PROGRAM ReadCP67
VAR
	
	ReadActLightLvlBoardroom :FB_DALIV2QueryActualLevel;  //Used to read back actual light lvl to correct dimmer on CP67 ask Plug top


	ADS_READ:ADSREAD;
	
	ADX_READ_DMXR:ADSREAD;
	ADX_READ_DMXG:ADSREAD;
	ADX_READ_DMXB:ADSREAD;
	
	DMX_Enable_READ:ADSREAD;
	
	HoldCP67BoardRoomLightsOn:BYTE;
	

	Sample		: BYTE;
	
	DMXRValues	:	ARRAY [0..7] OF BYTE;
	DMXGValues	:	ARRAY [0..7] OF BYTE;
	DMXBValues	:	ARRAY [0..7] OF BYTE;
	
	CP67_DMX_Enable	:	BOOL;
	
	FBDALIV2Dimmer1Switch : ARRAY [1..15] OF FB_DALIV2Dimmer1Switch;
	CASECP67BoardRoomLightsOn : INT;

END_VAR

sample := sample + 1;

FBDALIV2Dimmer1Switch[1](stCommandBuffer:= stCommandBuffer);
FBDALIV2Dimmer1Switch[2](stCommandBuffer:= stCommandBuffer);
ReadActLightLvlBoardroom(stCommandBuffer := stCommandBuffer , nActualLevel => BoardroomActualLightLvl ); 

IF CP67BoardRoomLightsOn <> HoldCP67BoardRoomLightsOn THEN
HoldCP67BoardRoomLightsOn := CP67BoardRoomLightsOn;
CASECP67BoardRoomLightsOn := 10;
END_IF

	CASE CASECP67BoardRoomLightsOn OF
		
	0: //Idle
	
	10:	FBDALIV2Dimmer1Switch[1].nDimmValue	:=  CP67BoardRoomLightsOn;
		FBDALIV2Dimmer1Switch[1].nAddr		:= 3;
		FBDALIV2Dimmer1Switch[1].eAddrType	:= 1;
			
		FBDALIV2Dimmer1Switch[2].nDimmValue	:=  CP67BoardRoomLightsOn; 
		FBDALIV2Dimmer1Switch[2].nAddr		:= 2; 
		FBDALIV2Dimmer1Switch[2].eAddrType	:= 1;
			
		CASECP67BoardRoomLightsOn			:= 20;	
			
	20:	IF  NOT FBDALIV2Dimmer1Switch[1].bBusy AND NOT FBDALIV2Dimmer1Switch[2].bBusy THEN
		CASECP67BoardRoomLightsOn 			:= 30;	

		ReadActLightLvlBoardroom.bStart		:= TRUE;
		ReadActLightLvlBoardroom.nAddr		:= 6;
		ReadActLightLvlBoardroom.eAddrType	:= 0;
		END_IF
	
	30:	IF NOT ReadActLightLvlBoardroom.bBusy THEN
		ReadActLightLvlBoardroom.bStart			:= FALSE;
		CASECP67BoardRoomLightsOn 				:= 0;
		
		END_IF
				
		
	END_CASE
		
	
	
	
(*// Send back actual light lvls for slider on CP67	
ReadActLightLvlBoardroom(
	bStart:= Sample.0, 
	nAddr:= 6, 
	eAddrType:= 0, 
	eCommandPriority:= , 
	bBusy=> , 
	bError=> , 
	nErrorId=> , 
	nActualLevel=> BoardroomActualLightLvl, 
	stCommandBuffer:= stCommandBuffer);	*)

(*
// DMX Values	
ADX_READ_DMXR(
	NETID:= '192.168.3.8.1.1', 
	PORT:= 851, 
	IDXGRP:= 16#4020, 
	IDXOFFS:= 1, 
	LEN:= 8, 
	DESTADDR:= ADR(DMXRValues), 
	READ:= Sample.0, 
	TMOUT:= T#2S, 
	BUSY=> , 
	ERR=> , 
	ERRID=> );
	
ADX_READ_DMXG(
	NETID:= '192.168.3.8.1.1', 
	PORT:= 851, 
	IDXGRP:= 16#4020, 
	IDXOFFS:= 9, 
	LEN:= 8, 
	DESTADDR:= ADR(DMXGValues), 
	READ:= Sample.0, 
	TMOUT:= T#2S, 
	BUSY=> , 
	ERR=> , 
	ERRID=> );
	
ADX_READ_DMXB(
	NETID:= '192.168.3.8.1.1', 
	PORT:= 851, 
	IDXGRP:= 16#4020, 
	IDXOFFS:= 17, 
	LEN:= 8, 
	DESTADDR:= ADR(DMXBValues), 
	READ:= Sample.0, 
	TMOUT:= T#2S, 
	BUSY=> , 
	ERR=> , 
	ERRID=> );
	
	
DMX_Enable_READ(
	NETID:= '192.168.3.8.1.1', 
	PORT:= 851, 
	IDXGRP:= 16#4020, 
	IDXOFFS:= 25, 
	LEN:= 1, 
	DESTADDR:= ADR(CP67_DMX_Enable), 
	READ:= Sample.0, 
	TMOUT:= T#2S, 
	BUSY=> , 
	ERR=> , 
	ERRID=> );
	*)

END_PROGRAM

(* stored: Version 1.1.0.1, ProductVersion 3.1.4024.12
   POU ReadCP67: Id {9520bf6c-b0a7-45ce-b025-02aba67bb34e}, SpecialFunc None *)
